{attribute 'GeneratedUsingTerminal: KL2004-0050'}
{attribute addProperty BoxType "KL2004-0050"}
{attribute addProperty Description ""}
{attribute addProperty Physics ""}
{attribute addProperty Id "Channel_1AT %Q*Channel_460B8C400Channel_2AT %Q*Channel_460B8C400Channel_3AT %Q*Channel_460B8C400Channel_4AT %Q*Channel_460B8C400Channel_5AT %Q*Channel_460B8C400Channel_6AT %Q*Channel_460B8C400Channel_7AT %Q*Channel_460B8C400Channel_8AT %Q*Channel_460B8C400Channel_9AT %Q*Channel_460B8C400Channel_10AT %Q*Channel_460B8C400Channel_11AT %Q*Channel_460B8C400Channel_12AT %Q*Channel_460B8C400Channel_13AT %Q*Channel_460B8C400Channel_14AT %Q*Channel_460B8C400Channel_15AT %Q*Channel_460B8C400Channel_16AT %Q*Channel_460B8C400Channel_17AT %Q*Channel_460B8C400Channel_18AT %Q*Channel_460B8C400Channel_19AT %Q*Channel_460B8C400Channel_20AT %Q*Channel_460B8C400Channel_21AT %Q*Channel_460B8C400Channel_22AT %Q*Channel_460B8C400Channel_23AT %Q*Channel_460B8C400Channel_24AT %Q*Channel_460B8C400Channel_25AT %Q*Channel_460B8C400Channel_26AT %Q*Channel_460B8C400Channel_27AT %Q*Channel_460B8C400Channel_28AT %Q*Channel_460B8C400Channel_29AT %Q*Channel_460B8C400Channel_30AT %Q*Channel_460B8C400Channel_31AT %Q*Channel_460B8C400Channel_32AT %Q*Channel_460B8C400"}
{attribute addProperty CRC "3472895434"}
{attribute addProperty Size "0"}
TYPE KL_CF002DCA :
STRUCT
	{attribute addProperty Name "Channel_1"}
	Channel_1 : Channel_460B8C40;
	{attribute addProperty Name "Channel_2"}
	Channel_2 : Channel_460B8C40;
	{attribute addProperty Name "Channel_3"}
	Channel_3 : Channel_460B8C40;
	{attribute addProperty Name "Channel_4"}
	Channel_4 : Channel_460B8C40;
	{attribute addProperty Name "Channel_5"}
	Channel_5 : Channel_460B8C40;
	{attribute addProperty Name "Channel_6"}
	Channel_6 : Channel_460B8C40;
	{attribute addProperty Name "Channel_7"}
	Channel_7 : Channel_460B8C40;
	{attribute addProperty Name "Channel_8"}
	Channel_8 : Channel_460B8C40;
	{attribute addProperty Name "Channel_9"}
	Channel_9 : Channel_460B8C40;
	{attribute addProperty Name "Channel_10"}
	Channel_10 : Channel_460B8C40;
	{attribute addProperty Name "Channel_11"}
	Channel_11 : Channel_460B8C40;
	{attribute addProperty Name "Channel_12"}
	Channel_12 : Channel_460B8C40;
	{attribute addProperty Name "Channel_13"}
	Channel_13 : Channel_460B8C40;
	{attribute addProperty Name "Channel_14"}
	Channel_14 : Channel_460B8C40;
	{attribute addProperty Name "Channel_15"}
	Channel_15 : Channel_460B8C40;
	{attribute addProperty Name "Channel_16"}
	Channel_16 : Channel_460B8C40;
	{attribute addProperty Name "Channel_17"}
	Channel_17 : Channel_460B8C40;
	{attribute addProperty Name "Channel_18"}
	Channel_18 : Channel_460B8C40;
	{attribute addProperty Name "Channel_19"}
	Channel_19 : Channel_460B8C40;
	{attribute addProperty Name "Channel_20"}
	Channel_20 : Channel_460B8C40;
	{attribute addProperty Name "Channel_21"}
	Channel_21 : Channel_460B8C40;
	{attribute addProperty Name "Channel_22"}
	Channel_22 : Channel_460B8C40;
	{attribute addProperty Name "Channel_23"}
	Channel_23 : Channel_460B8C40;
	{attribute addProperty Name "Channel_24"}
	Channel_24 : Channel_460B8C40;
	{attribute addProperty Name "Channel_25"}
	Channel_25 : Channel_460B8C40;
	{attribute addProperty Name "Channel_26"}
	Channel_26 : Channel_460B8C40;
	{attribute addProperty Name "Channel_27"}
	Channel_27 : Channel_460B8C40;
	{attribute addProperty Name "Channel_28"}
	Channel_28 : Channel_460B8C40;
	{attribute addProperty Name "Channel_29"}
	Channel_29 : Channel_460B8C40;
	{attribute addProperty Name "Channel_30"}
	Channel_30 : Channel_460B8C40;
	{attribute addProperty Name "Channel_31"}
	Channel_31 : Channel_460B8C40;
	{attribute addProperty Name "Channel_32"}
	Channel_32 : Channel_460B8C40;
END_STRUCT
END_TYPE

(* stored: Version 1.2.0.0, ProductVersion 3.1.4024.11
   DUT KL_CF002DCA: Id {fe9ededf-ea6d-4b41-9a7e-8399c99a1aa3} *)
